(* IEC 61131-3 sources: Std_PalletMover/Class/MQTTTopic_RetVals, 1 file *)

(* ---- MQTTTopic_RetVals.st ---- *)
(*!
<Class
	Name               = "MQTTTopic_RetVals"
	Revision           = "1.0"
	RealtimeTask       = "false"
	CyclicTask         = "false"
	BackgroundTask     = "false"
	Sigmatek           = "true"
	OSInterface        = "false"
	HighPriority       = "false"
	Automatic          = "false"
	UpdateMode         = "Prescan"
	SharedCommandTable = "true"
	Objectsize         = "(416,120)">
	<Channels>
		<Server Name="ClassSvr" Visualized="false" Initialize="false" WriteProtected="true" Retentive="false"/>
		<Server Name="udCRC" Visualized="false" Initialize="true" DefValue="-1" WriteProtected="false" Retentive="SRam"/>
	</Channels>
	<RevDoku>
		<Owner Company="Sigmatek"/>
		<Dokumentation Revision="1.0" Date="2020-03-04" Author="VelGer" Company="Sigmatek" Description="1. Initial Creation"/>
	</RevDoku>
</Class>
*)
MQTTTopic_RetVals : CLASS
  //Servers:
	ClassSvr 	: SvrChCmd_DINT;
	udCRC 	: SvrCh_UDINT;
  //Clients:
  //Variables:
  //Functions:
  //Tables:
	FUNCTION @STD
		VAR_OUTPUT
			ret_code	: CONFSTATES;
		END_VAR;
	FUNCTION GLOBAL TAB @CT_;
END_CLASS;
